DATA_BLOCK "InstRoboter"
{ S7_Optimized_Access := 'TRUE' }
VERSION : 0.1
NON_RETAIN
"Robot"

BEGIN

END_DATA_BLOCK

